RoboDK station: UR10-Robotiq.rdk

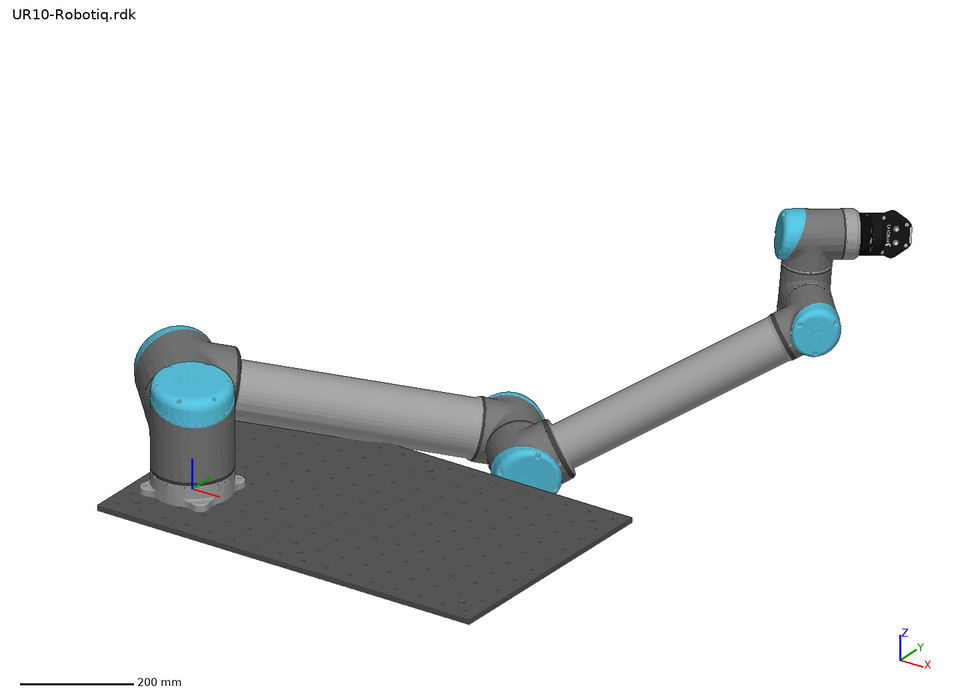
[picture v0: the station drawn from its stored meshes, robots at their saved joint values, targets as dots, program paths as lines]
Station UR10-Robotiq (saved by RoboDK 5.4.0). Poses are relative to the parent item; angles as X-Y-Z fixed-axis rotations.
  - frame UR10 Base at (0, 0, 0) mm
    - robot UR10: 6 axes, payload 10 kg, reach 1300 mm, repeatability 0.1 mm, weight 28.9 kg
        modified DH rows (alpha deg, a mm, theta deg, d mm): 0, 0, 0, 128; 90, 0, 180, 0; 0, 612.7, 0, 0; 0, 571.6, 0, 163.9; -90, 0, 0, 115.7; 90, 0, 180, 92.2
        joint limits [-360, -360, -360, -360, -360, -360] to [360, 360, 360, 360, 360, 360]; home [0, -90, -90, 0, 90, 0]; saved at [222.72, 13.753, -39.65, 210.375, 271.215, -99.046]
      - tool WRIST_CAMERA_20171116, TCP at (0, 0, 200) mm, size 75 x 87.5 x 22.4 mm, geometry from WRIST_CAMERA_20171116.STEP
      - robot RobotiQ 2F85: 1 axes, payload 5 kg
          joint limits [0] to [85]; home [85]; saved at [31.32]
      - frame RobotiQ 2F85 Base at (941.61, 1243.08, -3165.66) mm
  - object Plate-800x500-10mm v1 at (-100, -150, 0) mm, rotated rx 90 ry 0 rz 0 deg, size 800 x 10 x 500 mm, geometry from Plate-800x500-10mm v1.step
